Staubli VAL3: page_trajectory.dtx

num nIndex
num nKey = -1
public num nPage
num nRefresh = 2164.601
num nSelected
num nTime = 0.1
num nView
num nType
string sEvent = "hello"
string sEventImport
string sImport
public string sItems
string sList = "hello"
string sMenu[8]
  [0] = "Simulation"
  [4] = "Type"
  [5] = "Duplicate"
  [6] = "Delete"
  [7] = "New"
string sMenu8[8]
string sMenuUser[8]
string sMessage
bool bButton[8]
  [4] = true
  [5] = true
  [6] = true
  [7] = true
bool bLarge
num nIndexItem
num nOldIndex
bool bTrigger
num nClockStatus
bool bShowStatus
bool bMoveRelease
string sWorkingmode[8]
  [0] = "0 安全过度点 Joint"
  [1] = "1 Appro"
pointRx pPointTest[7]
  [0] = {fatherId=world[0]}
  [1] = {fatherId=world[0]}
  [2] = {fatherId=world[0]}
  [3] = {fatherId=world[0]}
  [4] = {fatherId=world[0]}
  [5] = {fatherId=world[0]}
  [6] = {fatherId=world[0]}
string sTrsfNum[8 6]
